FUNCTION_BLOCK FB_CylinderDoubleActing IMPLEMENTS ICylinder
VAR
	SolenoidA AT %Q* : BOOL;
	SolenoidB AT %Q* : BOOL;
END_VAR

METHOD Extend : BOOL
SolenoidA := TRUE;
SolenoidB := FALSE;
Extend	  := TRUE;
END_METHOD

METHOD Retract : BOOL
SolenoidA := FALSE;
SolenoidB := TRUE;
Retract	  := TRUE;
END_METHOD

END_FUNCTION_BLOCK

(* stored: Version 1.1.0.1, ProductVersion 3.1.4024.12
   POU FB_CylinderDoubleActing: Id {e79988e4-e59a-4ec8-94ee-4d878cd4b439}, SpecialFunc None
   Method Extend: Id {a0cbbcca-d7cf-4269-85d7-937dca0db2d9}
   Method Retract: Id {00a6b42e-fc0f-4b52-af30-c48ce772c915} *)
